FUNCTION_BLOCK FB_FallibleLREALMock IMPLEMENTS I_FallibleLREAL
VAR
    bError : BOOL;
    fVal : LREAL;
END_VAR

METHOD ClearError
END_METHOD

METHOD GetError : BOOL
GetError := THIS^.bError;
END_METHOD

METHOD GetErrorMsg : T_MaxString
END_METHOD

METHOD PUBLIC SetError
VAR_INPUT
    sMsg : T_MaxString;
END_VAR
THIS^.bError := TRUE;
END_METHOD

PROPERTY Val : LREAL
GET

Val := THIS^.fVal;
END_GET
SET
THIS^.fVal := Val;
END_SET
END_PROPERTY

END_FUNCTION_BLOCK

(* stored: Version 1.1.0.1, ProductVersion 3.1.4022.18
   POU FB_FallibleLREALMock: Id {fc0d4adc-5ab5-42f3-aed1-3f96b9aad2c8}, SpecialFunc None
   Method ClearError: Id {257abcd7-2766-4f1c-92bf-ac3f4824802a}
   Method GetError: Id {1db0c1f9-ea29-4eb4-b3c2-ed6d76aeeb6c}
   Method GetErrorMsg: Id {74cace86-ae75-47a5-9182-ceddc0340bcd}
   Method SetError: Id {aec07e5e-daa8-4bda-ba33-93ef3b5971b6}
   Property Val: Id {47717363-9808-4ba3-abcf-273c25c2c33e}
   Get Get: Id {c315ab54-4a35-41e3-a268-ba2f2abc5808}
   Set Set: Id {7926bd64-2e17-49c8-adc0-3a6d19fda8ac} *)
